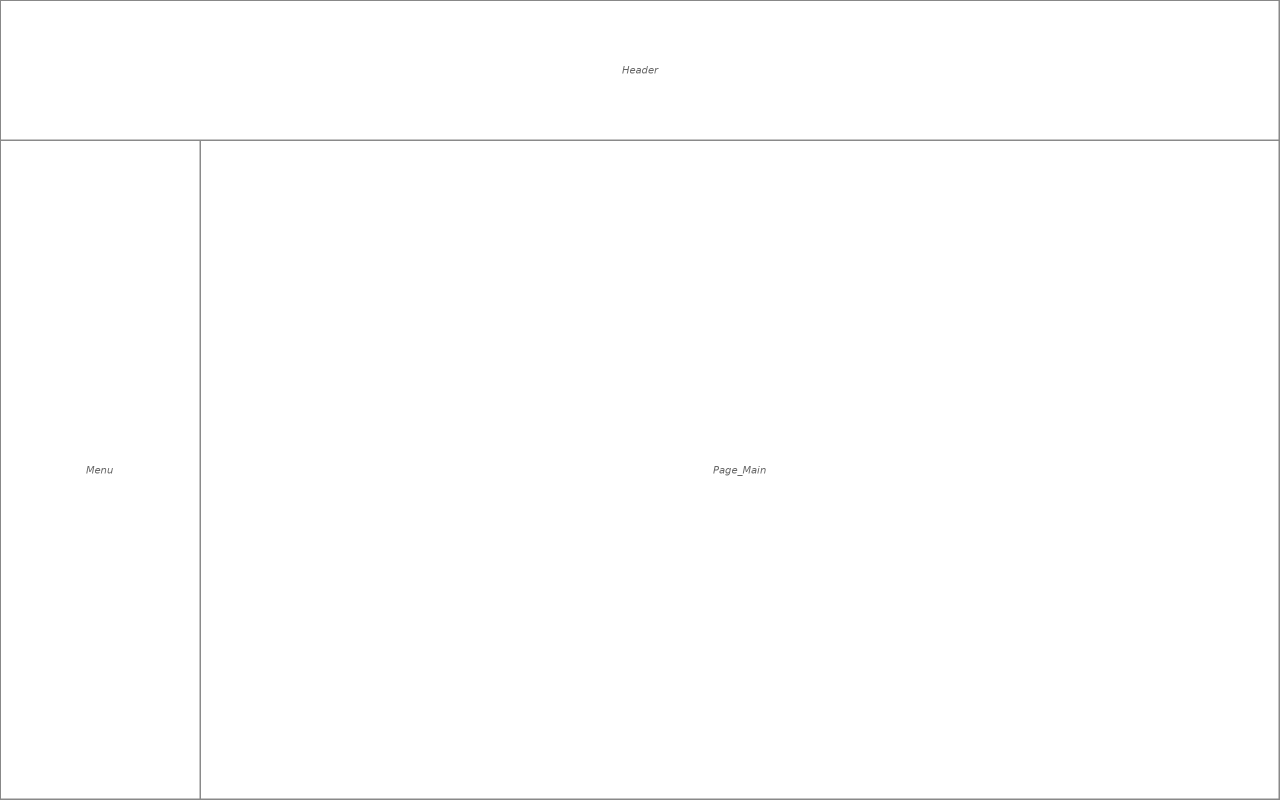
VISUALIZATION Main  // 1280x800
    Frame (0,140 200x660)
        shows Menu(i_itfVisuMenu := GVL_Visu.g_fbMenu)
    Frame (0,0 1280x140)
        shows Header()
    Frame (200,140 1080x660), frame switch variable: GVL_Visu.g_fbMenu.p_nPage
        shows Page_Main()
        shows Page_Infeed()
        shows Page_PackML()
        shows Page_Alarms()
END_VISUALIZATION

(* stored: Version 1.1.0.1, ProductVersion 3.1.4026.13
   Visu Main: Id {b1eb4e64-9153-40c9-9580-a92161dc9cb9} *)
